FUNCTION_BLOCK Sensor_4a20 (* Composite Function Block Type *)
  (* Standard: 61499-2 *)
  (* Version 0.0, 1/29/2026, Schneider Electric, template *)
  PACKAGE Hidryco.HidrycoLib;
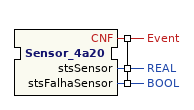
  EVENT_OUTPUT
    CNF WITH stsSensor, stsFalhaSensor;
  END_EVENT
  VAR_OUTPUT
    stsSensor : REAL;
    stsFalhaSensor : BOOL;
  END_VAR
  FBS
    FB1 : escalonamento;
    FB2 : alarmeHH_H_L_LL(modoAlarme := 1);
    IThis : Sensor_4a20_HMI(QI := TRUE);
    SYMLINKMULTIVARDST1 : SYMLINKMULTIVARDST_5A03F112CD5D470(QI := TRUE, NAME1 := '$${PATH}stsSensorBruto'); {SET_ATTRIBUTE(Configuration.GenericFBType.InterfaceParams, Runtime.System#I:=1;VALUE${I$}:INT)}
    plcStart1 : plcStart(Prio := 10);
  END_FBS
  EVENT_CONNECTIONS
    FB1.CNF TO FB2.E_ATUALIZA_ENTRADA;
    plcStart1.FIRST_INIT TO SYMLINKMULTIVARDST1.INIT;
    plcStart1.REDO_INIT TO SYMLINKMULTIVARDST1.INIT;
    SYMLINKMULTIVARDST1.CNF TO FB1.REQ;
    FB1.CNF TO CNF;
    SYMLINKMULTIVARDST1.INITO TO IThis.C9CE7FEC97FF63B7;
    FB1.CNF TO IThis.2DEB590422843D34;
    FB2.CNF TO IThis.71375A55927266AF;
    IThis.F2D08E9F122F71EC TO plcStart1.ACK_FIRST;
    IThis.A6B8B755362E8EC7 TO FB2.E_ATUALIZA_SETPOINTS;
    IThis.A6B8B755362E8EC7 TO FB1.E_AJUSTE_STP;
    IThis.8DBA3B6148BD206C TO FB1.E_RESET_FALHA;
    IThis.72E98372F71595E3 TO FB2.E_RESET_ALARMES;
  END_CONNECTIONS
  DATA_CONNECTIONS
    FB1.stsSensorEscalonado TO FB2.stsEntradaAlarme;
    SYMLINKMULTIVARDST1.VALUE1 TO FB1.stsSensorBruto;
    FB1.stsSensorEscalonado TO stsSensor;
    FB1.stsFalhaSensor TO stsFalhaSensor;
    FB1.stsSensorEscalonado TO IThis.C0ABCDF075E1A79D;
    FB1.stsFalhaSensor TO IThis.E9985E431FB89A02;
    FB2.stsAlarmeHH TO IThis.C82CA801D1092F6C;
    FB2.stsAlarmeH TO IThis.AE7C4A899B580B26;
    FB2.stsAlarmeL TO IThis.CD2C51A78C03C466;
    FB2.stsAlarmeLL TO IThis.1FB759DE167297C2;
    IThis.939069D94C475C89 TO FB2.stsSensorHabilitado;
    IThis.86A5D97104638E60 TO FB2.cmdHabilitaAlarmeHH;
    IThis.57577517CE80C66F TO FB2.cmdHabilitaAlarmeH;
    IThis.77B70C97887188C5 TO FB2.cmdHabilitaAlarmeL;
    IThis.62DA0CAC2BCB7CAE TO FB2.cmdHabilitaAlarmeLL;
    IThis.34F5DC7AAFC95566 TO FB1.stpRangeMaximo;
    IThis.76FB2D298BA4774E TO FB1.stpRangeMinimo;
    IThis.18DB3DA4763C63D TO FB2.stpTempoAlarmeHH;
    IThis.822C226C3EFAF836 TO FB2.stpTempoAlarmeH;
    IThis.61B311799E9F3DA2 TO FB2.stpTempoAlarmeL;
    IThis.71A70E331E6B2281 TO FB2.stpTempoAlarmeLL;
    IThis.656A4C528450D991 TO FB2.stpAlarmeHH;
    IThis.DDB0422C0CB760AD TO FB2.stpAlarmeH;
    IThis.AD1FE71FA411C38B TO FB2.stpAlarmeL;
    IThis.1CFB95872D4B3C1B TO FB2.stpAlarmeLL;
  END_CONNECTIONS
END_FUNCTION_BLOCK
